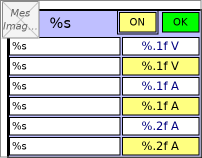
VISUALIZATION VISU_MARK3_PLUS  // 202x158
VAR_IN_OUT
	m_Input_IAD : BLOCK_MARK3_PLUS;
END_VAR
    Rectangle (7,9 195x149)
    Rectangle (162,12 37x20), "NOK", invisible if: (m_Input_IAD.IN_BUSSTAT) <> 0
    Rectangle (119,12 37x20), "OFF", invisible if: (m_Input_IAD.STATE_BEAM OR m_Input_IAD.STATE_BEAM_ON) <> 0
    Rectangle (162,12 37x20), "OK", invisible if: NOT m_Input_IAD.IN_BUSSTAT
    Rectangle (119,12 37x20), "ON", invisible if: NOT m_Input_IAD.STATE_BEAM AND NOT m_Input_IAD.STATE_BEAM_ON
    RoundedRectangle (9,37 111x18), "%s", text list: 'TextList_IAD', text index: 0
    RoundedRectangle (122,37 77x18), "%.1f V", text variable: m_Input_IAD.STATE_V_Anode
    RoundedRectangle (9,77 111x18), "%s", text list: 'TextList_IAD', text index: 1
    RoundedRectangle (122,77 77x18), "%.1f A", text variable: m_Input_IAD.STATE_I_Anode
    Rectangle (119,12 37x20), "ON", invisible if: (m_Input_IAD.STATE_BEAM_ON OR NOT m_Input_IAD.STATE_BEAM) <> 0
    Rectangle (7,12 107x22), "%s", text variable: m_Input_IAD.MNEMO
    Polyline (7,35)
    RoundedRectangle (9,57 111x18), "%s", invisible if: NOT Global_Variables.PRG_USER.ACTU_USER.MAINTENANCE OR NOT MACHINE.State_manu, text list: 'TextList_IAD', text index: 0
    RoundedRectangle (122,57 77x18), "%.1f V", text variable: m_Input_IAD.PRM_ANODE_VOLTAGE, invisible if: NOT Global_Variables.PRG_USER.ACTU_USER.MAINTENANCE OR NOT MACHINE.State_manu
        OnMouseDown: write the text variable via VisuDialogs.Numpad, min 0, max 300
    RoundedRectangle (9,97 111x18), "%s", invisible if: NOT Global_Variables.PRG_USER.ACTU_USER.MAINTENANCE OR NOT MACHINE.State_manu, text list: 'TextList_IAD', text index: 1
    RoundedRectangle (122,97 77x18), "%.1f A", text variable: m_Input_IAD.PRM_ANODE_CURRENT, invisible if: NOT Global_Variables.PRG_USER.ACTU_USER.MAINTENANCE OR NOT MACHINE.State_manu
        OnMouseDown: write the text variable via VisuDialogs.Numpad, min 0, max 15
    Rectangle (117,10 41x24), invisible if: NOT m_Input_IAD.BEAM.AUTOR_ON_IHM AND NOT m_Input_IAD.BEAM.AUTOR_OFF_IHM, input disabled if: ((NOT m_Input_IAD.BEAM.AUTOR_ON_IHM AND NOT m_Input_IAD.BEAM.AUTOR_OFF_IHM) OR NOT PRG_User.ACTU_USER.MAINTENANCE) <> 0
        OnMouseUp: execute { m_Input_IAD.BEAM.M_On:=(TRUE); }
    RoundedRectangle (9,117 111x18), "%s", text list: 'TextList_IAD', text index: 2
    RoundedRectangle (122,117 77x18), "%.2f A", text variable: m_Input_IAD.STATE_I_Neut
    RoundedRectangle (9,137 111x18), "%s", invisible if: NOT Global_Variables.PRG_USER.ACTU_USER.MAINTENANCE OR NOT MACHINE.State_manu, text list: 'TextList_IAD', text index: 2
    RoundedRectangle (122,137 77x18), "%.2f A", text variable: m_Input_IAD.PRM_NEUTRAL_CURRENT, invisible if: NOT Global_Variables.PRG_USER.ACTU_USER.MAINTENANCE OR NOT MACHINE.State_manu
        OnMouseDown: write the text variable via VisuDialogs.Numpad, min 0, max 1.86
    Image (2,1 37x37), invisible if: NOT m_Input_IAD.STATE_Nok, image: MesImages.warning
END_VISUALIZATION

(* stored: Version 1.1.0.1, ProductVersion 3.1.4024.10
   Visu VISU_MARK3_PLUS: Id {b5d73fee-4220-4103-8152-9324b092b5b5} *)
